PROGRAM PedestrianTrafficLight
VAR
	GreenTimerOn : BOOL := FALSE;
END_VAR

CASE GVL.StatusPedestrianLight OF

//Red Light
   0:
      GVL.PedestrianLightRed := TRUE;
      GVL.PedestrianLightGreen := FALSE;
	  
	  IF GVL.StatusCarLight = 2 THEN
		 GVL.StatusPedestrianLight := 1;
	  END_IF
	  
//Green light
   1:IF GVL.CarSensor THEN
	   GVL.StatusPedestrianLight := 2;
     ELSE
     GVL.PedestrianLightRed := FALSE;
     GVL.PedestrianLightGreen := TRUE;
	 END_IF
	 
// Waiting time for car	 
2:  GVL.TONPedestrianGreen(IN := TRUE , PT := T#10S);
	
    IF GVL.TONPedestrianGreen.ET >= T#5S THEN
       GVL.TONBlinkerTimer (IN := TRUE , PT := T#500MS );
       IF GVL.TONBlinkerTimer.Q THEN
          GVL.PedestrianLightGreen := NOT GVL.PedestrianLightGreen;
		  GVL.TONBlinkerTimer (IN := FALSE);
		  GVL.TONBlinkerTimer (IN := TRUE);
	   END_IF
	ELSE
		GVL.PedestrianLightGreen := TRUE;
    END_IF
	
    IF GVL.TONPedestrianGreen.Q THEN
	   GVL.StatusPedestrianLight := 0;
       GVL.TONPedestrianGreen (IN := FALSE);
	   GVL.TONBlinkerTimer (IN := FALSE);
	   GVL.PedestrianLightGreen := FALSE;
	END_IF
END_CASE

END_PROGRAM

(* stored: Version 1.1.0.1, ProductVersion 3.1.4024.12
   POU PedestrianTrafficLight: Id {fb27f1c4-8fe7-4552-9e6a-3e079d037577}, SpecialFunc None *)
